Staubli VAL3: writeSocket.pgx

program writeSocket(num handle_, string msg_)
  local num i
begin
  // write string to socket character by character
  for i=0 to (len(msg_)-1)
    sioSet(sSocket[handle_],asc(msg_,i))
  endFor
  sioSet(sSocket[handle_],13)
  sioSet(sSocket[handle_],10)
  if bDebug
    putln("writeStr: "+msg_)
  endIf
end
